// TIA Portal V20 export
DATA_BLOCK "DB_OPC_AxisManagement"   // DB105
// stored: InstanceOfName FB_OPC_AxisManagement, InstanceOfType FB
"FB_OPC_AxisManagement"
   // VAR
   //    sTeachButton : "FB_HmiKeysSignals";
   //    sAxisToTeachIndex { S7_SetPoint := 'True'} : DInt;
   //    sPositionToTeachIndex : DInt;
   //    sError { ExternalAccessible := 'False'; ExternalVisible := 'False'; ExternalWritable := 'False'} : Bool;
   //    sDone { ExternalAccessible := 'False'; ExternalVisible := 'False'; ExternalWritable := 'False'} : Bool;
   //    sState { ExternalAccessible := 'False'; ExternalVisible := 'False'; ExternalWritable := 'False'} : Word;
   //    sReadGUD_X_Load : "LBP_ReadGUD";
   //    sReadGUD_X_Unload { S7_SetPoint := 'True'} : "LBP_ReadGUD";
   //    sReadGUD_X_Blowing { S7_SetPoint := 'True'} : "LBP_ReadGUD";
   //    sReadGUD_Y_Load : "LBP_ReadGUD";
   //    sReadGUD_Y_Unload { S7_SetPoint := 'True'} : "LBP_ReadGUD";
   //    sReadGUD_Y_Blowing { S7_SetPoint := 'True'} : "LBP_ReadGUD";
   //    sReadGUD_B_Load : "LBP_ReadGUD";
   //    sReadGUD_B_Unload { S7_SetPoint := 'True'} : "LBP_ReadGUD";
   //    sReadGUD_B_Blowing { S7_SetPoint := 'True'} : "LBP_ReadGUD";
   //    sReadGUD_ZM_Safe { S7_SetPoint := 'True'} : "LBP_ReadGUD";
   //    sReadGUD_ZL_Safe { S7_SetPoint := 'True'} : "LBP_ReadGUD";
   //    sVarName { S7_SetPoint := 'True'} : String;
   //    sTON_On : TON_TIME;
   //    sTON_OFF { S7_SetPoint := 'True'} : TON_TIME;
   //    sPulseReadGUD { S7_SetPoint := 'True'} : Bool;
   //    sID : Int;
   // END_VAR
BEGIN
END_DATA_BLOCK
